(*
Interface for single-input controller toolbox components.

Implementors expose a write-only :attr:`Input` property. For components that
also produce an output signal, use :itf:`I_SisoComponent` instead.
*)
INTERFACE I_SiComponent

// Gets or sets the input to the component.
PROPERTY Input : LREAL
GET
END_GET
SET
END_SET
END_PROPERTY

END_INTERFACE

(* stored: Version 1.1.0.1, ProductVersion 3.1.4024.15
   Itf I_SiComponent: Id {7b82b91b-5b8f-4dcd-819c-0b83277c0b7a}
   Property Input: Id {687bf238-d9f7-4936-86a3-5ac32e13df89}
   Get Get: Id {654a203d-7616-4acf-a31d-2390624e1a0a}
   Set Set: Id {1ea30284-7813-46aa-bda5-7ff17b13e590} *)
